FUNCTION_BLOCK FB_ROB EXTENDS FB_Base IMPLEMENTS ITF_1_Robot, ITF_CommunicationModul

VAR_INPUT
	Skills: ARRAY[1..3] OF FB_Skill;
	SH: FB_SkillHandler;
END_VAR

VAR_INPUT
	ComConfig: ST_CommunicationConfig;

END_VAR


VAR_OUTPUT
	_inCollision: BOOL;
	 eConnectionState : eCommunicationState :=
        eCommunicationState.DISCONNECTED;
END_VAR
VAR
	    // ============================================================
    // Internal state
    // ============================================================

    _Connected : BOOL;
    _Busy : BOOL;


    _Command : STRING(1023);
    _CommandPending : BOOL;

    _ReconnectTimer : TON;
    _TimeoutTimer : TON;


    // Rising-edge detection
	
    _ExecuteConnect : BOOL;
    _ExecuteDisconnect : BOOL;
    _ExecuteCommand : BOOL;

    _LastCommand : STRING(1023);
	
	
	_enabled: BOOL;
	_mode: eMode;
	_locked: BOOL;
	
	velovr: BOOL;
	velfact: REAL;
	
	DBClient: FB_PostgreSQLClient;
	

END_VAR


VAR
    // =========================================================
    // Communication state
    // =========================================================

   

    xConnectRequest : BOOL := FALSE;
    xDisconnectRequest : BOOL := FALSE;

    // One-shot execute signals
    xSocketConnectExecute : BOOL := FALSE;
    xSocketCloseExecute : BOOL := FALSE;


    fbSocketConnect : FB_SocketConnect;
    fbSocketClose : FB_SocketClose;

    hSocket : T_HSOCKET;


    SocketErrorId : UDINT := 0;
END_VAR

//State Machine
ComMachine();
DBClient();

METHOD ComMachine : BOOL
VAR_INPUT
END_VAR
CASE eConnectionState OF


    // =========================================================
    // DISCONNECTED
    // =========================================================

    eCommunicationState.DISCONNECTED:

       _connected := FALSE;


        // Make sure socket handle is cleared
//         hSocket


        // -----------------------------------------------------
        // Connect requested
        // -----------------------------------------------------

        IF xConnectRequest THEN

            xConnectRequest := FALSE;

            // Clear previous errors
            Error := FALSE;
            ErrorId := 0;
            SocketErrorId := 0;

            // Start FB_SocketConnect
            xSocketConnectExecute := TRUE;

            eConnectionState :=
                eCommunicationState.CONNECTING;

        END_IF;


    // =========================================================
    // CONNECTING
    // =========================================================

    eCommunicationState.CONNECTING:

        _connected := FALSE;
        


        // -----------------------------------------------------
        // Execute FB_SocketConnect
        // -----------------------------------------------------

        fbSocketConnect(
            sSrvNetId := '',
            sRemoteHost := ComConfig.sIpAddress,
            nRemotePort := ComConfig.nPort,
            bExecute := xSocketConnectExecute,
            tTimeout := ComConfig.tTimeout
        );


        // Execute must only be TRUE for one cycle
        xSocketConnectExecute := FALSE;


        // -----------------------------------------------------
        // Connection successful
        // -----------------------------------------------------

        IF NOT fbSocketConnect.bBusy
            AND NOT fbSocketConnect.bError
//             AND (fbSocketConnect.hSocket <> 0)
        THEN

            hSocket :=
                fbSocketConnect.hSocket;

            _connected := TRUE;
    

            Error := FALSE;
            ErrorId := 0;
            SocketErrorId := 0;

            eConnectionState :=
                eCommunicationState.CONNECTED;

        END_IF;


        // -----------------------------------------------------
        // Connection failed
        // -----------------------------------------------------

        IF NOT fbSocketConnect.bBusy
            AND fbSocketConnect.bError
        THEN

            _connected := FALSE;

            Error := TRUE;

            SocketErrorId :=
                fbSocketConnect.nErrId;

            ErrorId :=
                fbSocketConnect.nErrId;

//             hSocket := 0;

            eConnectionState :=
                eCommunicationState.ERROR;

        END_IF;


    // =========================================================
    // CONNECTED
    // =========================================================

    eCommunicationState.CONNECTED:

        _connected := TRUE;



        // -----------------------------------------------------
        // Disconnect requested
        // -----------------------------------------------------

        IF xDisconnectRequest THEN

            xDisconnectRequest := FALSE;


            // Start socket close
            xSocketCloseExecute := TRUE;

            eConnectionState :=
                eCommunicationState.DISCONNECTING;

        END_IF;


    // =========================================================
    // DISCONNECTING
    // =========================================================

    eCommunicationState.DISCONNECTING:

        _connected := FALSE;


        // -----------------------------------------------------
        // Execute FB_SocketClose
        // -----------------------------------------------------

        fbSocketClose(
            sSrvNetId := '',
            hSocket := hSocket,
            bExecute := xSocketCloseExecute,
            tTimeout := ComConfig.tTimeout
        );


        // Execute only for one cycle
        xSocketCloseExecute := FALSE;


        // -----------------------------------------------------
        // Socket closed successfully
        // -----------------------------------------------------

        IF NOT fbSocketClose.bBusy
            AND NOT fbSocketClose.bError
        THEN

            _connected := FALSE;


//             hSocket := 0;

            eConnectionState :=
                eCommunicationState.DISCONNECTED;

        END_IF;


        // -----------------------------------------------------
        // Socket close failed
        // -----------------------------------------------------

        IF NOT fbSocketClose.bBusy
            AND fbSocketClose.bError
        THEN

            _connected := FALSE;


            Error := TRUE;

            SocketErrorId :=
                fbSocketClose.nErrId;

            ErrorId :=
                fbSocketClose.nErrId;

            // The socket should no longer be used
//             hSocket := 0;

            eConnectionState :=
                eCommunicationState.ERROR;

        END_IF;


    // =========================================================
    // ERROR
    // =========================================================

    eCommunicationState.ERROR:

        _connected := FALSE;
        // -----------------------------------------------------
        // Do not attempt to use the socket after an error
        // -----------------------------------------------------

//         hSocket := 0;


        // -----------------------------------------------------
        // A new connection request can recover from the error
        // -----------------------------------------------------

        IF xConnectRequest THEN

            xConnectRequest := FALSE;

            Error := FALSE;
            ErrorId := 0;
            SocketErrorId := 0;

            xSocketConnectExecute := TRUE;

            eConnectionState :=
                eCommunicationState.CONNECTING;

        END_IF;


END_CASE;
END_METHOD

{warning 'Add method implementation '}
METHOD Connect : BOOL

Connect := FALSE;

// Already connected
IF eConnectionState = eCommunicationState.CONNECTED THEN
    Connect := TRUE;
    RETURN;
END_IF;

// Already trying to connect
IF eConnectionState = eCommunicationState.CONNECTING THEN
    Connect := TRUE;
    RETURN;
END_IF;

// Don't accept a new connection while disconnecting
IF eConnectionState = eCommunicationState.DISCONNECTING THEN
    RETURN;
END_IF;

// Validate address
IF LEN(ComConfig.sIpAddress) = 0 THEN
    Error := TRUE;
//     ErrorId := 16#1001;
    RETURN;
END_IF;

// Validate port
IF ComConfig.nPort = 0 THEN
    Error := TRUE;
//     ErrorId := 16#1002;
    RETURN;
END_IF;

// Clear previous error
Error := FALSE;
ErrorId := 0;

// Request connection
xConnectRequest := TRUE;

Connect := TRUE;
END_METHOD

{warning 'Add property implementation'}
PROPERTY Connected : BOOL
GET
Connected:=_connected;
END_GET
END_PROPERTY

{warning 'Add method implementation '}
METHOD Disconnect : BOOL
END_METHOD

{warning 'Add method implementation '}
METHOD M_AUTO : BOOL
_mode:=eMode.Automatic;
END_METHOD

{warning 'Add method implementation '}
METHOD M_Disable : BOOL
_enabled:=FALSE;
super^.Deactivate();
END_METHOD

{warning 'Add method implementation '}
METHOD M_DisableVelocityOverride : BOOL
velovr:=False;
END_METHOD

{warning 'Add method implementation '}
METHOD M_Enable : BOOL
_enabled:=TRUE;
END_METHOD

{warning 'Add method implementation '}
METHOD M_EnableVelocityOverride : BOOL
velovr:=True;
END_METHOD

{warning 'Add method implementation '}
METHOD M_EStop : BOOL
END_METHOD

{warning 'Add method implementation '}
METHOD M_MAN : BOOL
_mode:=eMode.Manual;
END_METHOD

{warning 'Add method implementation '}
METHOD MC_ChangeSpeedOverride : INT
VAR_INPUT
	factor	: REAL;
END_VAR
velfact:=factor;
END_METHOD

METHOD onActivate : BOOL
// ---- Init ----
transitionresult:=eResult.None;



// ---- Change ----

// _mode:= eMode.Automatic;




// ---- Check ----
transitionresult := eResult.SUCCESS;


// ---- Change State ----
IF transitionresult= eResult.SUCCESS THEN
	State:=eState.Active;
ELSIF transitionresult= eResult.FAILURE THEN
	State:=eState.Inactive;
ELSIF transitionresult= eResult.ERROR THEN
	State:=eState.ErrorProcessing;
ELSE
	ADSLOGSTR(ADSLOG_MSGTYPE_WARN,'Transitionresult from onActivate is None','');
END_IF
END_METHOD

METHOD onCleanup : BOOL
// ---- Init ----
transitionresult:=eResult.None;



// ---- Change ----

_mode:= eMode.Manual;




// ---- Check ----
transitionresult := eResult.SUCCESS;


// ---- Change State ----
IF transitionresult= eResult.SUCCESS THEN
	State:=eState.Unconfigured;
ELSIF transitionresult= eResult.FAILURE THEN
	ADSLOGSTR(ADSLOG_MSGTYPE_WARN,'Transitionresult from onCleanup is FAILURE ','');
ELSIF transitionresult= eResult.ERROR THEN
	State:=eState.ErrorProcessing;
ELSE
	ADSLOGSTR(ADSLOG_MSGTYPE_WARN,'Transitionresult from onCleanup is NONE','');
END_IF
END_METHOD

METHOD onConfigure : BOOL
// ---- Init ----
transitionresult:=eResult.None;



// ---- Change ----

_mode:= eMode.Manual;




// ---- Check ----
transitionresult := eResult.SUCCESS;


// ---- Change State ----
IF transitionresult= eResult.SUCCESS THEN
	State:=eState.Inactive;
ELSIF transitionresult= eResult.FAILURE THEN
	State:=eState.Unconfigured;
ELSIF transitionresult= eResult.ERROR THEN
	State:=eState.ErrorProcessing;
ELSE
	ADSLOGSTR(ADSLOG_MSGTYPE_WARN,'Transitionresult from onConfigure is None','');
END_IF
END_METHOD

METHOD onDeactivate : BOOL
// ---- Init ----
transitionresult:=eResult.None;



// ---- Change ----

_mode:= eMode.Manual;




// ---- Check ----
transitionresult := eResult.SUCCESS;


// ---- Change State ----
IF transitionresult= eResult.SUCCESS THEN
	State:=eState.Inactive;
ELSIF transitionresult= eResult.FAILURE THEN
	ADSLOGSTR(ADSLOG_MSGTYPE_WARN,'Transitionresult from onDeactivate is FAILURE','');
ELSIF transitionresult= eResult.ERROR THEN
	State:=eState.ErrorProcessing;
ELSE
	ADSLOGSTR(ADSLOG_MSGTYPE_WARN,'Transitionresult from onDeactivate is None','');
END_IF
END_METHOD

METHOD onError : BOOL
// ---- Init ----
transitionresult:=eResult.None;



// ---- Change ----

_mode:= eMode.Manual;




// ---- Check ----
transitionresult := eResult.SUCCESS;


// ---- Change State ----
IF transitionresult= eResult.SUCCESS THEN
	State:=eState.Unconfigured;
ELSIF transitionresult= eResult.FAILURE THEN
	State:=eState.Finalized;
ELSIF transitionresult= eResult.ERROR THEN
	ADSLOGSTR(ADSLOG_MSGTYPE_WARN,'Transitionresult from onError is Error','');
ELSE
	ADSLOGSTR(ADSLOG_MSGTYPE_WARN,'Transitionresult from onError is None','');
END_IF
END_METHOD

METHOD onShutdown : BOOL
// ---- Init ----
transitionresult:=eResult.None;



// ---- Change ----

_mode:= eMode.Manual;




// ---- Check ----
transitionresult := eResult.SUCCESS;


// ---- Change State ----
IF transitionresult= eResult.SUCCESS THEN
	State:=eState.Finalized;
ELSIF transitionresult= eResult.FAILURE THEN
	ADSLOGSTR(ADSLOG_MSGTYPE_WARN,'Transitionresult from onShutdown is FAILURE','');
ELSIF transitionresult= eResult.ERROR THEN
	State:=eState.ErrorProcessing;
ELSE
	ADSLOGSTR(ADSLOG_MSGTYPE_WARN,'Transitionresult from onShutdown is None','');
END_IF
END_METHOD

{warning 'Add property implementation'}
PROPERTY P_isInCollision : BOOL
GET
P_isInCollision:=_inCollision;
END_GET
END_PROPERTY

{warning 'Add property implementation'}
PROPERTY P_JogSpeed : LREAL
GET
END_GET
SET
END_SET
END_PROPERTY

{warning 'Add property implementation'}
PROPERTY P_RobotIsMoving : BOOL
GET
END_GET
END_PROPERTY

{warning 'Add property implementation'}
PROPERTY P_RobotIsReady : BOOL
GET
END_GET
END_PROPERTY

{warning 'Add method implementation '}
METHOD ResetConnection : BOOL
END_METHOD

END_FUNCTION_BLOCK

(* stored: Version 1.1.0.1, ProductVersion 3.1.4026.18
   POU FB_ROB: Id {7ce28b50-28f8-4d4c-bb25-1006bf064637}, SpecialFunc None
   Folder Communication: Id {482fc868-908c-498f-adb6-41c2da0d8c6c}
   Folder StateControl: Id {306f9b72-2cb2-4dec-88a3-0a1776eb8cb9}
   Method ComMachine: Id {f49a5e24-a4a9-4b80-8d0f-86db7d255ee2}
   Method Connect: Id {047fe0b6-5747-4791-80bd-12650d215bd4}
   Property Connected: Id {80fca5f5-8709-4982-a384-df957ec0f13e}
   Get Get: Id {99f48d79-5a32-4dfc-8ac6-28f7e421e088}
   Method Disconnect: Id {ee0b7b31-ec5f-4f91-978c-fcaa048156f8}
   Method M_AUTO: Id {a36cbff6-922e-4670-8cae-63446b6e1765}
   Method M_Disable: Id {bbb8a1cb-19df-48a2-aa34-15efcd08818d}
   Method M_DisableVelocityOverride: Id {ee13b86f-55fa-4515-ac1d-c418ff59ec19}
   Method M_Enable: Id {3bb80d4c-ff29-49a1-abc5-c8b4d3120296}
   Method M_EnableVelocityOverride: Id {1ca0163b-6260-47a4-b242-d72534327ea7}
   Method M_EStop: Id {ff1c583d-626a-4142-b727-591a7a8cf9e6}
   Method M_MAN: Id {3ea33c07-baa7-444c-a0bc-e71071e519dd}
   Method MC_ChangeSpeedOverride: Id {a5e39256-a687-447d-8a2a-a95ea9e40d2e}
   Method onActivate: Id {92a2cf27-c6ee-447f-b5b4-e372093c0834}
   Method onCleanup: Id {b8d25f1a-bd56-4d52-bf77-294e7c965601}
   Method onConfigure: Id {da5be059-6955-4a6d-bdaf-05a0e2dc60bb}
   Method onDeactivate: Id {9cfadd55-1f96-401b-82a9-c49bdb0b9d71}
   Method onError: Id {af5714ff-685b-4718-92d7-e4e00300345c}
   Method onShutdown: Id {54edc0cd-8c64-49fa-9d9a-b9e92650f21c}
   Property P_isInCollision: Id {8eea56b9-50ca-4510-b567-db19e3eca5c7}
   Get Get: Id {885867df-c0d3-4443-aec9-8d2b982d76c4}
   Property P_JogSpeed: Id {b02ce28c-7dc7-4355-aadb-75f0e04880fa}
   Get Get: Id {5422baec-3cfa-49de-a9e5-c204b5dc3b85}
   Set Set: Id {70edccef-4005-4ebc-8367-68039a4d1e15}
   Property P_RobotIsMoving: Id {d73761d6-28bd-445a-ae23-6297821e885b}
   Get Get: Id {afd258f0-1b48-45c8-895f-cafec57170be}
   Property P_RobotIsReady: Id {749d199f-9e7a-4d77-b560-89090e6f1785}
   Get Get: Id {69a643b8-e941-4372-aaf0-4d36068ddfee}
   Method ResetConnection: Id {1825ac35-9b96-4ce0-86aa-50b35c933301} *)
